// TIA Portal V20 export
VAR_GLOBAL   // PLC tag table "Default tag table"
   adat1 AT %IW0 : Int;
   adat2 AT %IW2 : Int;
   adat3 AT %IW4 : Int;
   adat4 AT %IW6 : Int;
   adat5 AT %IW8 : Int;
   adat6 AT %IW10 : Int;
   adat7 AT %IW12 : Int;
   adat8 AT %IW14 : Word;
END_VAR
